Staubli VAL3: ListPop.pgx

program ListPop(string x_sS (dimensions=1))
begin
  switch sLanguge
    case "English"
      call ListPopE(x_sS)
    break
    case "Chinese"
      call ListPopC(x_sS)
    break
  endSwitch
end
